// TIA Portal V16 export
// export: Created 2022-01-12T14:34:28.1373866Z, ExportSetting WithDefaults, DisplayName Totally Integrated Automation Portal, DisplayVersion V16 Update 4, DisplayName TIA Portal Version Control Interface, DisplayVersion V16 Update 2, DisplayName TIA Portal Openness, DisplayVersion V16 Update 4, DisplayName STEP 7 Professional, DisplayVersion V16 Update 4, DisplayName STEP 7 Safety, DisplayVersion V16, DisplayName WinCC Professional, DisplayVersion V16 Update 4
TYPE "typSygnały"
// stored: IsFailsafeCompliant false
   STRUCT
      S : Array[1..50] of Bool;   // sygnał
   END_STRUCT;
   // // S[1] : CIP1
   // // S[2] : CIP2
   // // S[3] : CIP3
   // // S[4] : TANK_CIP
   // // S[5] : READY1
   // // S[6] : READY2
   // // S[7] : READY3
   // // S[8] : READY4
   // // S[9] : CONF1
   // // S[10] : CONF2
   // // S[11] : CONF3
   // // S[12] : CONF4
   // // S[13] : ERR
   // // S[14] : PULLOUT1
   // // S[15] : PULLOUT2
   // // S[16] : PULLOUT3
   // // S[17] : WATER1
   // // S[18] : WATER2
   // // S[19] : WATER3
   // // S[20] : OUT1
   // // S[21] : OUT2
   // // S[22] : OUT3
   // // S[23] : CONNECT1
   // // S[24] : CONNECT2
   // // S[25] : CONNECT3
   // // S[26] : WHEY
   // // S[27] : AG
   // // S[28] : PUMP
   // // S[29] : FLIP
   // // S[30] : RUNNING
   // // S[31] : FEED
   // // S[32] : START
   // // S[33] : REMOTE
   // // S[34] : RINSING
   // // S[35] : ERR
   // // S[36] : OUT
   // // S[37] : ZS01
   // // S[38] : ZS02
   // // S[39] : ZS03
   // // S[40] : ZS04
   // // S[41] : ZS05
END_TYPE
